(* CODESYS project xlh_dc_motor_00_01.project
   Description: Receives some incoming messages and echoes them with CAN-ID +1
   Company: 3S - Smart Software Solutions GmbH
   Version: 1.0.0.0
   Title: CAN Bus API Example
   Author: 3S - Smart Software Solutions GmbH

Project tree, tasks and I/O mapping:
  xLH_base : CODESYS Control for Raspberry Pi 64 SL, CODESYS, order no. 2302000009, version 4.18.0.0
    application app
      libraries: Standard, 3.5.18.0 (System); Util, 3.5.21.0 (System); VisuDialogs, * (System); Memory, * (3S - Smart Software Solutions GmbH); CmpBitmapPool, * (System); CAN API, 1.0.0.4 (CODESYS); MemoryUtils, * (3S - Smart Software Solutions GmbH); CAA CiA 405, 4.3.0.0 (CODESYS); xLH Control Systems, 0.1 (xemax ag)
      task MAIN_TASK (cyclic, interval 10 ms, priority 1) calls RET_DCM, io
      task VISU_TASK (cyclic, interval 100 ms, priority 31) calls VisuElems.Visu_Prg
      trace Trace_Switch (task MAIN_TASK): MAIN.diEncoderPosition, MAIN.fSpeed, MAIN.fCurrentMa
      program io [ST]
      program RET_DCM [CFC]
      visualisation VISU_RET_DCM
      function block Dynamik [ST]: Dynamiktyp
      data type eDynamiktyp
    SoftMotion General Axis Pool
      a_axis : SM_Drive_PosControl, CODESYS, order no. 1805, version 4.18.0.0
          settings: wDriveID = 4; dwRatioTechUnitsDenom = 101846; iRatioTechUnitsNum = -125; eRampType = 1; fSWMaxVelocity = 50; fSWMaxAcceleration = 100; fSWMaxDeceleration = 100; fSWMaxJerk = 1000; fSWLimitNegative = -1000.0; ScalingIncs = 814768; ScalingUnits = 1000; InvertDirection = TRUE; IsLinearMotor = TRUE; MaximumOutputVelocityInt = 40738; MinimumOutputVelocityInt = -40738; Kp = 0.05; MaxFollowingError = 5.0; EnableFollowingErrorCheck = TRUE; DeadTime = 3.0
      x_axis : SM_Drive_PosControl, CODESYS, order no. 1805, version 4.18.0.0
          settings: dwRatioTechUnitsDenom = 101846; iRatioTechUnitsNum = 125; eRampType = 1; fSWMaxVelocity = 50; fSWMaxAcceleration = 100; fSWMaxDeceleration = 100; fSWMaxJerk = 1000; fSWLimitNegative = -1000; ScalingIncs = 814768; ScalingUnits = 1000; IsLinearMotor = TRUE; MaximumOutputVelocityInt = 40738; MinimumOutputVelocityInt = -40738; Kp = 0.05; MaxFollowingError = 5.0; EnableFollowingErrorCheck = TRUE; DeadTime = 3.0
      y_axis : SM_Drive_PosControl, CODESYS, order no. 1805, version 4.18.0.0
          settings: wDriveID = 2; dwRatioTechUnitsDenom = 101846; iRatioTechUnitsNum = 125; eRampType = 1; fSWMaxVelocity = 50; fSWMaxAcceleration = 100; fSWMaxDeceleration = 100; fSWMaxJerk = 1000; fSWLimitNegative = -1000; ScalingIncs = 814768; ScalingUnits = 1000; IsLinearMotor = TRUE; MaximumOutputVelocityInt = 40738; MinimumOutputVelocityInt = -40738; Kp = 0.05; MaxFollowingError = 5.0; EnableFollowingErrorCheck = TRUE; DeadTime = 3.0
      z_axis : SM_Drive_PosControl, CODESYS, order no. 1805, version 4.18.0.0
          settings: wDriveID = 3; dwRatioTechUnitsDenom = 101846; iRatioTechUnitsNum = 125; eRampType = 1; fSWMaxVelocity = 50; fSWMaxAcceleration = 100; fSWMaxDeceleration = 100; fSWMaxJerk = 1000; fSWLimitNegative = -1000; ScalingIncs = 814768; ScalingUnits = 1000; IsLinearMotor = TRUE; MaximumOutputVelocityInt = 40738; MinimumOutputVelocityInt = -40738; Kp = 0.05; MaxFollowingError = 5.0; EnableFollowingErrorCheck = TRUE; DeadTime = 3.0
    GPIOs_A_B : GPIOs B+/Pi2, CODESYS, version 4.18.0.0
        unmapped channels: digital inputs (GPIO0..GPIO31), digital outputs (GPIO0..GPIO31)
    Onewire
    Camera device
      <Leer>
    SPI
    I²C
    CANbus : CANbus, CODESYS, version 4.3.0.0
        settings: Baudrate = 1000 kbit/s
      CANopen_Manager : CANopen_Manager, CODESYS, version 4.3.0.0
          settings: ConfigVersion = 50659584
        xlh_dc_motor : xlh_dc_motor, xemax ag, order no. 0, version Revision=16#00000001, FileVersion=1.0
            settings: NODEIDSAVED = 1; SDO Timeout = 1000000; PDO_Autoconfig = FALSE; EXPERTSETTINGS = FALSE; PDO 16#1400.COBID = 16#00000201; Process by CANopenManager = TRUE; PDO 16#1800.COBID = 16#00000181; Process by CANopenManager = TRUE; Control.Subindex = 16#01; PWM Duty Cycle.Subindex = 16#02; Position.Subindex = 16#01; dt per Increment.Subindex = 16#02; Current.Subindex = 16#01; SDO List.Set COB-ID sync.Index = 16#1005; SDO List.Set COB-ID sync.Subindex = 16#00; SDO List.Set COB-ID sync.Value = 16#00000080; SDO List.Set COB-ID sync.Size = 32; SDO List.Set COB-ID sync.AbortIfError = FALSE; SDO List.Set COB-ID sync.JumpToLine = FALSE; SDO List.Set COB-ID sync.Line = 0; SDO List.Set communication cycle period.Index = 16#1006; SDO List.Set communication cycle period.Subindex = 16#00; SDO List.Set communication cycle period.Value = 16#00000000; SDO List.Set communication cycle period.Size = 32; SDO List.Set communication cycle period.AbortIfError = FALSE; SDO List.Set communication cycle period.JumpToLine = FALSE; SDO List.Set communication cycle period.Line = 0; SDO List.Set Guardtime.Index = 16#100C; SDO List.Set Guardtime.Subindex = 16#00; SDO List.Set Guardtime.Value = 16#000000C8; SDO List.Set Guardtime.Size = 16; SDO List.Set Guardtime.AbortIfError = FALSE; SDO List.Set Guardtime.JumpToLine = FALSE; SDO List.Set Guardtime.Line = 0; SDO List.Set Lifetime.Index = 16#100D; SDO List.Set Lifetime.Subindex = 16#00; SDO List.Set Lifetime.Value = 16#00000003; SDO List.Set Lifetime.Size = 8; SDO List.Set Lifetime.AbortIfError = FALSE; SDO List.Set Lifetime.JumpToLine = FALSE;
              SDO List.Set Lifetime.Line = 0; SDO List.Set Heartbeat Consumer.Index = 16#1016; SDO List.Set Heartbeat Consumer.Subindex = 16#01; SDO List.Set Heartbeat Consumer.Value = 0; SDO List.Set Heartbeat Consumer.Size = 32; SDO List.Set Heartbeat Consumer.AbortIfError = FALSE; SDO List.Set Heartbeat Consumer.JumpToLine = FALSE; SDO List.Set Heartbeat Consumer.Line = 0; SDO List.Disable PDO.Index = 16#1400; SDO List.Disable PDO.Subindex = 16#01; SDO List.Disable PDO.Value = 16#80000201; SDO List.Disable PDO.Size = 32; SDO List.Disable PDO.AbortIfError = FALSE; SDO List.Disable PDO.JumpToLine = FALSE; SDO List.Disable PDO.Line = 0; SDO List.Set transmission type.Index = 16#1400; SDO List.Set transmission type.Subindex = 16#02; SDO List.Set transmission type.Value = 16#FF; SDO List.Set transmission type.Size = 8; SDO List.Set transmission type.AbortIfError = FALSE; SDO List.Set transmission type.JumpToLine = FALSE; SDO List.Set transmission type.Line = 0; SDO List.Set and enable COB-ID.Index = 16#1400; SDO List.Set and enable COB-ID.Subindex = 16#01; SDO List.Set and enable COB-ID.Value = 16#00000201; SDO List.Set and enable COB-ID.Size = 32; SDO List.Set and enable COB-ID.AbortIfError = FALSE; SDO List.Set and enable COB-ID.JumpToLine = FALSE; SDO List.Set and enable COB-ID.Line = 0; SDO List.Disable PDO.Index = 16#1800; SDO List.Disable PDO.Subindex = 16#01; SDO List.Disable PDO.Value = 16#80000181; SDO List.Disable PDO.Size = 32; SDO List.Disable PDO.AbortIfError = FALSE; SDO List.Disable PDO.JumpToLine = FALSE; SDO List.Disable PDO.Line = 0; SDO List.Set transmission type.Index = 16#1800; SDO List.Set transmission type.Subindex = 16#02; SDO List.Set transmission type.Value = 16#FF; SDO List.Set transmission type.Size = 8;
              SDO List.Set transmission type.AbortIfError = FALSE; SDO List.Set transmission type.JumpToLine = FALSE; SDO List.Set transmission type.Line = 0; SDO List.Set inhibit time.Index = 16#1800; SDO List.Set inhibit time.Subindex = 16#03; SDO List.Set inhibit time.Value = 16#0000; SDO List.Set inhibit time.Size = 16; SDO List.Set inhibit time.AbortIfError = FALSE; SDO List.Set inhibit time.JumpToLine = FALSE; SDO List.Set inhibit time.Line = 0; SDO List.Set event time.Index = 16#1800; SDO List.Set event time.Subindex = 16#05; SDO List.Set event time.Value = 16#0000; SDO List.Set event time.Size = 16; SDO List.Set event time.AbortIfError = FALSE; SDO List.Set event time.JumpToLine = FALSE; SDO List.Set event time.Line = 0; SDO List.Set and enable COB-ID.Index = 16#1800; SDO List.Set and enable COB-ID.Subindex = 16#01; SDO List.Set and enable COB-ID.Value = 16#00000181; SDO List.Set and enable COB-ID.Size = 32; SDO List.Set and enable COB-ID.AbortIfError = FALSE; SDO List.Set and enable COB-ID.JumpToLine = FALSE; SDO List.Set and enable COB-ID.Line = 0; ConfigVersion = 50659584
            output app.io.bMotorCcw : BOOL  // Control.Bit0
            output app.io.bMotorCw : BOOL  // Control.Bit1
            output app.io.uiMotorSpeed : UINT  // PWM Duty Cycle
            input  app.io.diEncoderPosition : DINT  // Position
            input  app.io.iEncoderDtInc : INT  // dt per Increment
            input  app.io.uiCurrent : UINT  // Current
            unmapped channels: Control
  libraries: VisuSymbols, 4.5.0.0 (System); DepictorBase, 1.2.0.0 (CODESYS)
  text list GlobalTextList
  5ce3da45-db07-42e7-a21c-a00fff4ed8f6|C:\Users\phe\Downloads\Musterloesung_FUP.PNG
*)

// xLH_base/app/eDynamiktyp
{attribute 'qualified_only'}
{attribute 'strict'}
TYPE eDynamiktyp :
(
	Linear := 1,
	Quadratisch := 2
)INT;
END_TYPE

// xLH_base/app/RET_DCM
PROGRAM RET_DCM

VAR
	
	bENA_M1: BOOL := FALSE; // Freigabe M1
	bENA_M2: BOOL := FALSE; // Freigabe M2
	signalgeno_Y: Signalgenerator := (eTyp := eSignalform.OFFSET ,rOffset := 0.0, rAmplitude := 15.0, rFrequenz := 0.1, bRauschen := FALSE, rRauschenVerstaerkung := 1.0);	

	bRE_DrehzahlAktiv: BOOL; // Freigabe Drehzahl-Regler
	Regler_Drehzahl: Regler := (eTyp := eReglertyp.PI, rKr := 15.0, rTn := 0.25, rTv := 0.5, rTvz := 0.015, rYlim_max := 100.0, rYlim_min := 0.0, bEnable_AWU := TRUE);
	
	bRE_AWUAktiv: BOOL; // Aktiv AWU Drehzahl-Regler
	bAWU_UL_Aktiv: BOOL;
	bAWU_LL_Aktiv: BOOL;
	
	signalgeno_W_Drehzahl: Signalgenerator := (eTyp := eSignalform.RECHTECK ,rOffset := 2.5, rAmplitude := 0.5, rFrequenz := 0.2, bRauschen := FALSE, rRauschenVerstaerkung := 1.0);
	rW_f: REAL;
	rE_f: REAL;
	rY_f: REAL;  // vor Linearisierung
	rY_f_lin: REAL;  // nach Linearisierung
	rY_f_dynamik: REAL;  // nach Dynamik
	rX_f: REAL;
	
	// LOGGER
	bLoggerRunning: BOOL := FALSE;
	rLoggerTime_Drehzahl: REAL := 5;
	Logger_Drehzahl: Logger_;
	bENA_Linearisierung: BOOL;
	Linearisierung: Kennlinie := (bAktiviert := FALSE, bSpiegelungXgY := FALSE,
		arXin := [0.0, 0.1, 0.2, 0.3, 57.43, 72.9, 83.87, 91.94, 97.42, 100.0, 100.0],
		arYin := [0.0, 10.0, 20.0, 30.0, 40.0, 50.0, 60.0, 70.0, 80.0, 90.0, 100.0]);

END_VAR
VAR // added by the converter: edge detectors and wires of the graphical bodies
    _w1, _w2, _w3, _w4, _w5 : ANY;
END_VAR

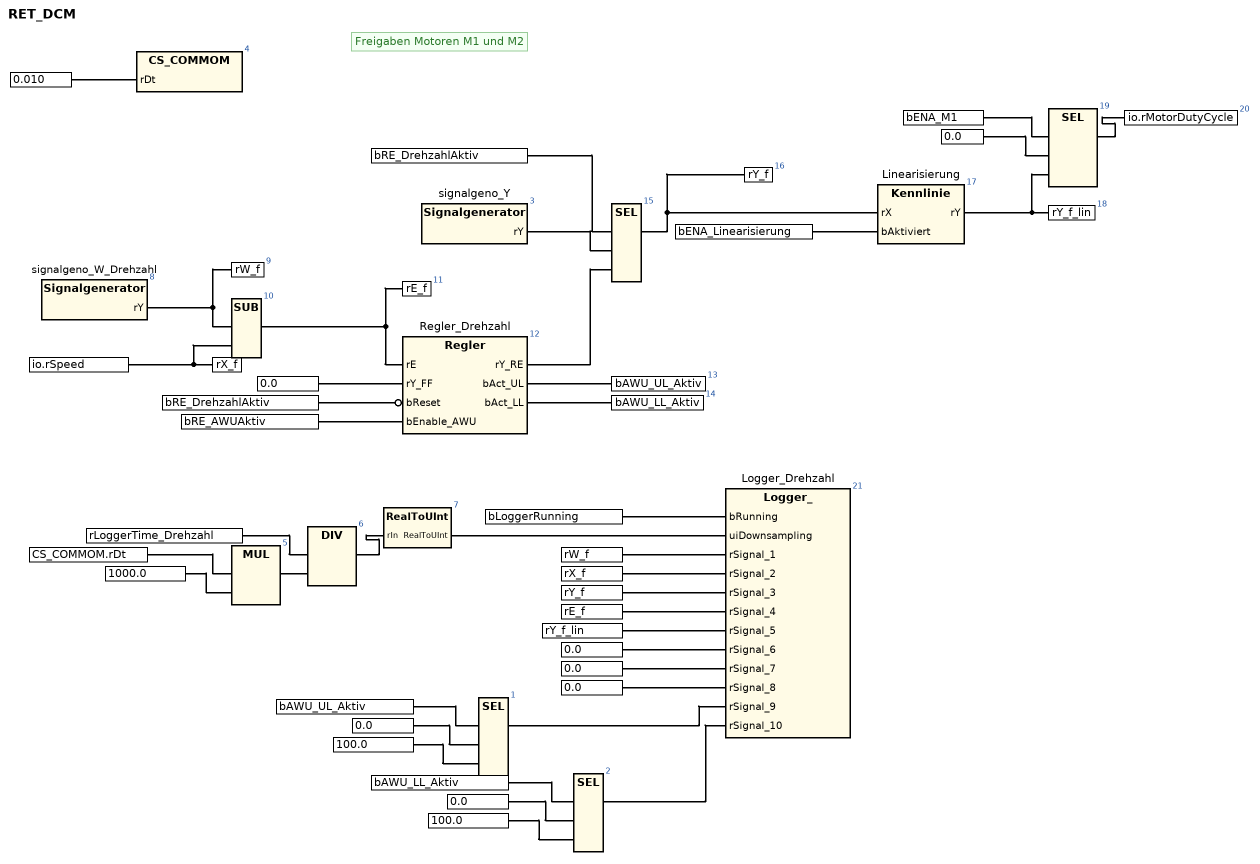
rX_f := io.rSpeed;
_w1 := SEL(bAWU_UL_Aktiv, 0.0, 100.0);
_w2 := SEL(bAWU_LL_Aktiv, 0.0, 100.0);
signalgeno_Y(); // Signalgenerator
// Freigaben Motoren M1 und M2
CS_COMMOM(rDt := 0.010);
_w3 := RealToUInt(rIn := rLoggerTime_Drehzahl / (CS_COMMOM.rDt * 1000.0));
signalgeno_W_Drehzahl(); // Signalgenerator
rW_f := signalgeno_W_Drehzahl.rY;
_w4 := signalgeno_W_Drehzahl.rY - io.rSpeed;
rE_f := _w4;
Regler_Drehzahl(rE := _w4, rY_FF := 0.0, bReset := NOT bRE_DrehzahlAktiv, bEnable_AWU := bRE_AWUAktiv); // Regler
bAWU_UL_Aktiv := Regler_Drehzahl.bAct_UL;
bAWU_LL_Aktiv := Regler_Drehzahl.bAct_LL;
_w5 := SEL(bRE_DrehzahlAktiv, signalgeno_Y.rY, Regler_Drehzahl.rY_RE);
rY_f := _w5;
Linearisierung(rX := _w5, bAktiviert := bENA_Linearisierung); // Kennlinie
rY_f_lin := Linearisierung.rY;
io.rMotorDutyCycle := SEL(bENA_M1, 0.0, Linearisierung.rY);
Logger_Drehzahl(
    bRunning := bLoggerRunning,
    uiDownsampling := _w3,
    rSignal_1 := rW_f,
    rSignal_2 := rX_f,
    rSignal_3 := rY_f,
    rSignal_4 := rE_f,
    rSignal_5 := rY_f_lin,
    rSignal_6 := 0.0,
    rSignal_7 := 0.0,
    rSignal_8 := 0.0,
    rSignal_9 := _w1,
    rSignal_10 := _w2); // Logger_

END_PROGRAM

// xLH_base/app/io
PROGRAM io
VAR_INPUT
	diEncoderPosition: DINT;
	iEncoderDtInc: INT;
	uiCurrent: UINT;
	rMotorDutyCycle: real;
END_VAR
VAR_OUTPUT
	bMotorCw: BOOL;
	bMotorCcw: BOOL;
	uiMotorSpeed: UINT;
	rSpeed: REAL;
	rCurrentMa: REAL;
	// FixMe: Vereinfachung
	bEna_Motor_quadratisch: BOOL := FALSE;
	rSkalierung: REAL := 100.0;
	bEna_Motoren_Dynamik: BOOL := FALSE;
	rZeitkonstante: REAL := 0.1;
END_VAR
VAR
		// Charakteristika Motor 
	// Stationäre Kennlinie
	Motoren_dynamik_stationaer: Dynamik := (rScalierung:= 100.0, iTyp:= 1);
	// Dynamik
	Motoren_dynamik_dynamisch: PT2 := (rK := 1.0, rT1:= 0.01, rT2:= 0.01);
	rY_1: REAL;
	rY_2: REAL;
	rSpeedTemp: REAL;
	fbPt2: PT2:= (rK:=1.0, rT1:= 0.040, rT2:= 0.040);
END_VAR

rCurrentMa := TO_REAL(uiCurrent) / 10.0;

// Encoder 20 Inc/turn
// gear ratio 1 / 36
// 1s = 1000000us
// Nominator = 1000000/(20*36) = 1388.88
IF iEncoderDtInc <> 0 THEN
	rSpeedTemp := 1388.88 / TO_REAL(iEncoderDtInc) ;
ELSE
	rSpeedTemp := 0.0;
END_IF
fbPt2(rX:=rSpeedTemp, rY=>rSpeed);


IF rMotorDutyCycle >= 0.0 THEN
	bMotorCw := TRUE;
	bMotorCcw := FALSE;
ELSE
	bMotorCw := FALSE;
	bMotorCcw := FALSE;
END_IF

// Einkopplung Charakteristik Motor stationär und dynamisch
// Stationäre Kennlinie
IF bEna_Motor_quadratisch THEN
	Motoren_dynamik_stationaer(rYin:=rMotorDutyCycle, rScalierung:=rSkalierung, iTyp:=2, rYout=>rY_1);
ELSE
	Motoren_dynamik_stationaer(rYin:=rMotorDutyCycle, rScalierung:=rSkalierung, iTyp:=1, rYout=>rY_1);
END_IF
// Dynamik
IF bEna_Motoren_Dynamik THEN
	Motoren_dynamik_dynamisch(rX:=rY_1, rT1:= rZeitkonstante, rT2:= rZeitkonstante, rY=>rY_2);
ELSE
	rY_2 := rY_1;
END_IF


uiMotorSpeed := REAL_TO_UINT(LIMIT(0.0, ABS(rY_2 * 450.0), 45000));
//uiMotorSpeed := REAL_TO_UINT(LIMIT(0.0, ABS(rMotorDutyCycle * 450.0), 45000)); 
//uiMotorSpeed := TO_UINT(ABS(rMotorDutyCycle) * 655.35);

END_PROGRAM

// xLH_base/app/Dynamik
FUNCTION_BLOCK Dynamik
VAR_INPUT
	rYin: REAL;
	rScalierung: REAL;
	eTyp:  eDynamiktyp;
	iTyp: INT;
END_VAR
VAR_OUTPUT
	rYout: REAL;
END_VAR
VAR
	rY_in: REAL;
	bLinear: BOOL;
	bQuadratisch: BOOL;
END_VAR

 

// Normierung
IF rScalierung > 0.0 THEN
	rY_in := rYin / rScalierung;
ELSE
	rY_in := rYin / 1.0;
END_IF

// Typ zuordnen -> später via Funktionsblock in der Lib
IF iTyp = 1 THEN
	rYout := rY_in;
ELSIF iTyp = 2 THEN
	rYout := rY_in * rY_in;
ELSE
	rYout := rY_in;
END_IF

// Ausgang setzen, abhängig vom Vorzeichen
IF rY_in >= 0.0 THEN
	rYout := rYout * rScalierung;
ELSE
	rYout := rYout * rScalierung * -1.0;
END_IF


// Dynamiktyp zuordnen
//IF bLinear THEN
//	rYout := rY_in;
//ELSIF bQuadratisch THEN
//	rYout := rY_in * rY_in;
//END_IF

ACTION Dynamiktyp:
// Auswahl möglicher Konfigurationen
CASE eTyp OF
	eDynamiktyp.Linear:
	 	bLinear := TRUE;
		bQuadratisch := FALSE;
	eDynamiktyp.Quadratisch:
		bLinear := FALSE;
		bQuadratisch := TRUE;
			
END_CASE
END_ACTION

END_FUNCTION_BLOCK

// xLH_base/app/VISU_RET_DCM
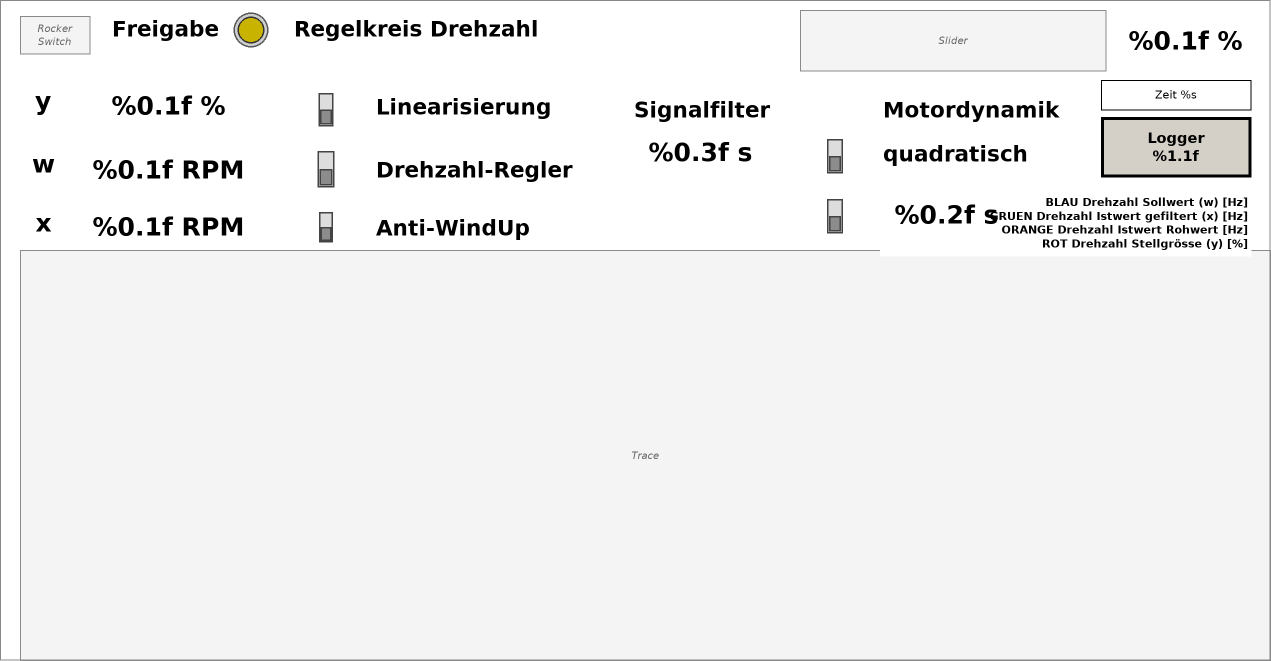
VISUALIZATION VISU_RET_DCM  // 1271x661
    Slider (800,10 306x61), variable: io.rMotorDutyCycle, scale -100..100
    Rectangle (1105,10 161x61), "%0.1f %", text variable: io.rMotorDutyCycle
    Rectangle (1101,80 150x30), "Zeit %s", text variable: RET_DCM.rLoggerTime_Drehzahl
        OnMouseDown: write the text variable via Default, min 5, max 7200
    Rectangle (1101,117 150x60), "Logger %1.1f", text variable: RET_DCM.logger_Drehzahl.rActIndexProzent, colour toggle: RET_DCM.bLoggerRunning
        OnMouseClick: execute {
            IF RET_DCM.Logger_Drehzahl.bRunning = FALSE THEN
            	RET_DCM.Logger_Drehzahl.iStateLogger := 1;
            	RET_DCM.Logger_Drehzahl.rActIndexProzent := 0.0;
            	RET_DCM.Logger_Drehzahl.bRunning := TRUE;
            ELSE
            	RET_DCM.Logger_Drehzahl.iStateLogger := 0;
            	RET_DCM.Logger_Drehzahl.rActIndexProzent := 0.0;
            	RET_DCM.Logger_Drehzahl.bRunning := FALSE;
            END_IF
        }
    Rectangle (291,10 310x38), "Regelkreis Drehzahl"
    Trace (20,250 1251x411)
    Rectangle (880,190 371x66), "BLAU Drehzahl Sollwert (w) [Hz] GRUEN Drehzahl Istwert gefiltert (x) [Hz] ORANGE Drehzahl Istwert Rohwert [Hz] ROT Drehzahl Stellgrösse (y) [%]"
    Rectangle (72,75 193x61), "%0.1f %", text variable: RET_DCM.rY_f
    Rectangle (20,80 47x41), "y"
        OnMouseClick:  Dialog=Dialog_Signalgenerator_Y, OpenModal=True, PositionX=200, PositionY=100
    Rectangle (20,141 47x45), "w"
        OnMouseClick:  Dialog=Dialog_Signalgenerator_W_Drehzahl, OpenModal=True, PositionX=100, PositionY=100
    Rectangle (72,139 193x61), "%0.1f RPM", text variable: RET_DCM.rW_f
    Rectangle (373,151 197x38), "Drehzahl-Regler"
        OnMouseClick:  Dialog=Dialog_Regler_Drehzahl, OpenModal=True, PositionX=100, PositionY=100
    DipSwitch (291,151 70x36), variable: RET_DCM.bRE_DrehzahlAktiv, behaviour: TOGGLE, style: Switch-DipSwitch-Gray
    Rectangle (373,88 197x38), "Linearisierung"
        OnMouseClick:  Dialog=Dialog_Linearisierung_Drehzahl, OpenModal=True, PositionX=100, PositionY=100
    Rectangle (72,196 193x61), "%0.1f RPM", text variable: RET_DCM.rX_f
    Rectangle (20,200 47x45), "x"
    DipSwitch (291,93 70x33), variable: RET_DCM.bENA_Linearisierung, behaviour: TOGGLE, style: Switch-DipSwitch-Gray
    DipSwitch (291,212 70x30), variable: RET_DCM.bRE_AWUAktiv, behaviour: TOGGLE, style: Switch-DipSwitch-Gray
    Rectangle (373,209 197x38), "Anti-WindUp"
    Rectangle (850,184 193x61), "%0.2f s", text variable: io.rZeitkonstante
        OnMouseClick: write the text variable via Default, min 0.01, max 10.00
    DipSwitch (800,139 70x34), variable: io.bEna_Motor_quadratisch, behaviour: TOGGLE, style: Switch-DipSwitch-Gray
    Rectangle (109,10 112x38), "Freigabe"
        OnMouseClick:  Dialog=Dialog_Linearisierung_Drehzahl, OpenModal=True, PositionX=100, PositionY=100
    RockerSwitch (20,16 70x38), variable: RET_DCM.bENA_M1, behaviour: TOGGLE, style: Switch-RockerSwitch-Gray
    Rectangle (880,91 197x38), "Motordynamik"
        OnMouseClick:  Dialog=Dialog_Linearisierung_Drehzahl, OpenModal=True, PositionX=100, PositionY=100
    Rectangle (880,136 197x38), "linear", invisible if: io.bEna_Motor_quadratisch
        OnMouseClick:  Dialog=Dialog_Linearisierung_Drehzahl, OpenModal=True, PositionX=100, PositionY=100
    Rectangle (880,135 197x38), "quadratisch", invisible if: not io.bEna_Motor_quadratisch
        OnMouseClick:  Dialog=Dialog_Linearisierung_Drehzahl, OpenModal=True, PositionX=100, PositionY=100
    Lamp1 (231,10 40x40), variable: RET_DCM.bENA_M1, style: Lamp-Lamp1-Yellow
    Rectangle (631,129 139x46), "%0.3f s", text variable: io.fbPt2.rT1
        OnMouseClick: write the text variable via Default, min 0.005, max 1.000
    DipSwitch (800,199 70x34), variable: io.bEna_Motoren_Dynamik, behaviour: TOGGLE, style: Switch-DipSwitch-Gray
    Rectangle (631,91 147x38), "Signalfilter"
        OnMouseClick:  Dialog=Dialog_Linearisierung_Drehzahl, OpenModal=True, PositionX=100, PositionY=100
END_VISUALIZATION
